TYPE ST_OperationVars_Grid:
STRUCT
	b_SyncClose							: BOOL;
END_STRUCT
END_TYPE

(* stored: Version 1.1.0.1, ProductVersion 3.1.4026.18
   DUT ST_OperationVars_Grid: Id {b3af3c02-c451-4e76-8f68-fe8d6201e230} *)
